// TIA Portal V16 export
// export: Created 2023-03-29T11:04:30.790865Z, ExportSetting WithDefaults, DisplayName Totally Integrated Automation Portal, DisplayVersion V16 Update 6, DisplayName TIA Portal Version Control Interface, DisplayVersion V16 Update 2, DisplayName TIA Portal Openness, DisplayVersion V16 Update 6, DisplayName STEP 7 Professional, DisplayVersion V16 Update 6, DisplayName STEP 7 Safety, DisplayVersion V16, DisplayName WinCC Advanced, DisplayVersion V16 Update 6
FUNCTION_BLOCK "Kontrola przeciążenia falownika"   // FB17, LAD
TITLE = Control Current Overload
{ S7_Optimized_Access := 'TRUE' }
AUTHOR : rtecmer
VERSION : 0.1
// Kontrola przeciążenia invertera KDN M25 M27
// stored: AutoNumber true, IsIECCheckEnabled false, IsRetainMemResEnabled false, MemoryReserve 500, SetENOAutomatically false, UDAEnableTagReadback false
BEGIN

REGION Network 1: Ustawienie wartości granicznej
   // Nastawa dopuszczalnego prądu invertera. Znacznik M10 zastosowany w celach serwisowych. Wybór ograniczenia z edytowanego z HMI lub z nastaw czytanych z falownika.
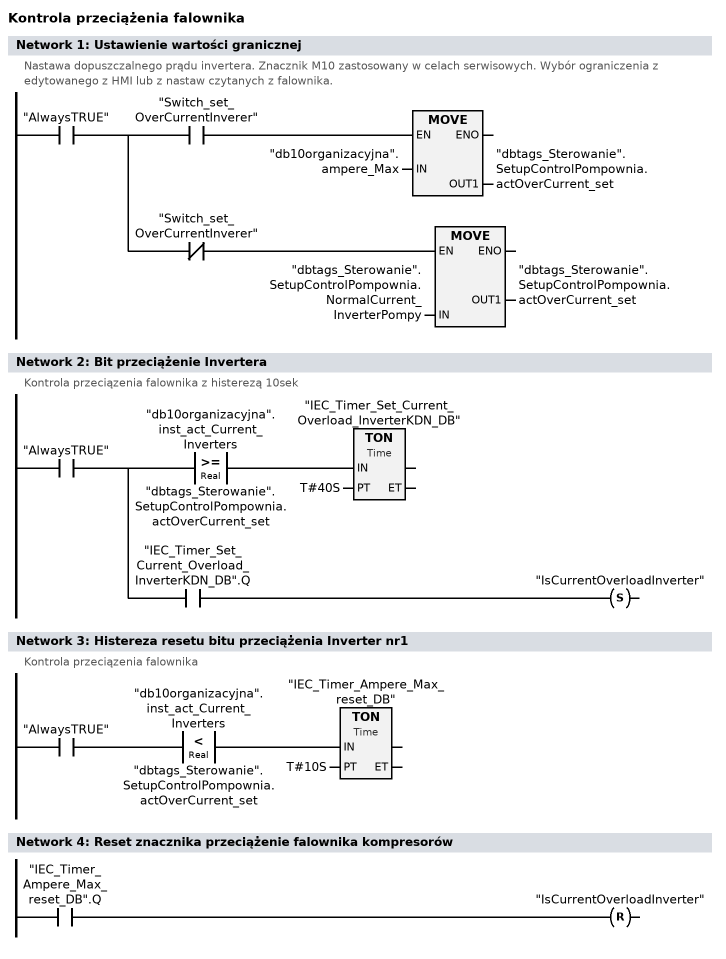
   RUNG wire#powerrail
      Contact( "AlwaysTRUE" )
      wire#w1
      Contact( "Switch_set_OverCurrentInverer" )
      Move(in := "db10organizacyjna".ampere_Max, out1 => "dbtags_Sterowanie".SetupControlPompownia.actOverCurrent_set)
   END_RUNG
   RUNG wire#w1
      I_Contact( "Switch_set_OverCurrentInverer" )
      Move(in := "dbtags_Sterowanie".SetupControlPompownia.NormalCurrent_InverterPompy, out1 => "dbtags_Sterowanie".SetupControlPompownia.actOverCurrent_set)
   END_RUNG
   // the same network as SCL:
   IF "AlwaysTRUE" AND "Switch_set_OverCurrentInverer" THEN
       "dbtags_Sterowanie".SetupControlPompownia.actOverCurrent_set := "db10organizacyjna".ampere_Max;
   END_IF;
   IF "AlwaysTRUE" AND NOT "Switch_set_OverCurrentInverer" THEN
       "dbtags_Sterowanie".SetupControlPompownia.actOverCurrent_set := "dbtags_Sterowanie".SetupControlPompownia.NormalCurrent_InverterPompy;
   END_IF;
END_REGION

REGION Network 2: Bit przeciążenie Invertera
   // Kontrola przeciązenia falownika z histerezą 10sek
   RUNG wire#powerrail
      Contact( "AlwaysTRUE" )
      wire#w1
      { S7_Templates := "SrcType := Real" } GE_Contact(in1 := "db10organizacyjna".inst_act_Current_Inverters, in2 := "dbtags_Sterowanie".SetupControlPompownia.actOverCurrent_set)
      { S7_Templates := "time_type := Time" } "IEC_Timer_Set_Current_Overload_InverterKDN_DB".TON(pt := T#40S, et =>)
   END_RUNG
   RUNG wire#w1
      Contact( "IEC_Timer_Set_Current_Overload_InverterKDN_DB".Q )
      S_Coil( "IsCurrentOverloadInverter" )
   END_RUNG
   // the same network as SCL:
   "IEC_Timer_Set_Current_Overload_InverterKDN_DB".TON(IN := "AlwaysTRUE" AND ("db10organizacyjna".inst_act_Current_Inverters >= "dbtags_Sterowanie".SetupControlPompownia.actOverCurrent_set),
                           PT := T#40S);
   IF "AlwaysTRUE" AND "IEC_Timer_Set_Current_Overload_InverterKDN_DB".Q THEN
       "IsCurrentOverloadInverter" := TRUE;
   END_IF;
END_REGION

REGION Network 3: Histereza resetu bitu przeciążenia Inverter nr1
   // Kontrola przeciązenia falownika
   RUNG wire#powerrail
      Contact( "AlwaysTRUE" )
      { S7_Templates := "SrcType := Real" } LT_Contact(in1 := "db10organizacyjna".inst_act_Current_Inverters, in2 := "dbtags_Sterowanie".SetupControlPompownia.actOverCurrent_set)
      { S7_Templates := "time_type := Time" } "IEC_Timer_Ampere_Max_reset_DB".TON(pt := T#10S, et =>)
   END_RUNG
   // the same network as SCL:
   "IEC_Timer_Ampere_Max_reset_DB".TON(IN := "AlwaysTRUE" AND ("db10organizacyjna".inst_act_Current_Inverters < "dbtags_Sterowanie".SetupControlPompownia.actOverCurrent_set),
                           PT := T#10S);
END_REGION

REGION Network 4: Reset znacznika przeciążenie falownika kompresorów
   RUNG wire#powerrail
      Contact( "IEC_Timer_Ampere_Max_reset_DB".Q )
      R_Coil( "IsCurrentOverloadInverter" )
   END_RUNG
   // the same network as SCL:
   IF "IEC_Timer_Ampere_Max_reset_DB".Q THEN "IsCurrentOverloadInverter" := FALSE; END_IF;
END_REGION
END_FUNCTION_BLOCK
